PROGRAM MAIN
VAR
END_VAR

END_PROGRAM

(* stored: Version 1.1.0.1
   POU MAIN: Id {a814c2dd-c1f5-4ba6-a0dd-2b94a9e246f0} *)
